TYPE SJH108IonizerConfig EXTENDS DeviceConfiguration :
STRUCT
	{attribute 'OPC.UA.DA' := '0'}
	IonizerAlarm : ARRAY [0..IonizerConst.NUMBER_ALARMS] OF IonizerAlarm;
END_STRUCT
END_TYPE

(* stored: Version 1.1.0.1, ProductVersion 3.1.4024.12
   DUT SJH108IonizerConfig: Id {f83f0867-41a9-45ee-9bd8-fb7572ce683f} *)
